// TIA Portal project "separating station" (V17)
// Vorlageprojekt für das Buch mit Zielsystem S7-1200

(* hardware
DEVICE "S7-1200-Station_1"  S7-1200 Station
   slot 0: "Baugruppenträger_0"  Rack  V1.0
   slot 1: "PLC_1"  CPU 1211C DC/DC/DC  6ES7 211-1AE40-0XB0  V4.1
*)

// ===== PLC "PLC_1"  CPU 1211C DC/DC/DC =====

VAR_GLOBAL   // PLC tag table "Standard-Variablentabelle"
   "senz 1" AT %I0.0 : Bool;
   "push 1 f" AT %I0.1 : Bool;
   "push 1 b" AT %I0.2 : Bool;
   "at push 1 exit" AT %I0.3 : Bool;
   "push 2 f" AT %I0.5 : Bool;
   "push 2 b" AT %I0.6 : Bool;
   "at push 2 exit" AT %I0.7 : Bool;
   "start" AT %I1.0 : Bool;
   "reset" AT %I1.1 : Bool;
   "stop" AT %I1.2 : Bool;
   "e stop" AT %I1.3 : Bool;
   "FACTORY io run" AT %I1.4 : Bool;
   "vs 1" AT %ID30 : DInt;
   "vs2" AT %ID34 : DInt;
   "entry conv 1" AT %Q0.0 : Bool;
   "pusher 1" AT %Q0.1 : Bool;
   "conv 1" AT %Q0.2 : Bool;
   "entry conv 2" AT %Q0.3 : Bool;
   "pusher 2" AT %Q0.4 : Bool;
   "conv 2" AT %Q0.5 : Bool;
   "start light" AT %Q0.6 : Bool;
   "reset light" AT %Q0.7 : Bool;
   "stop light" AT %Q1.0 : Bool;
   "count 2" AT %QD30 : DInt;
   "count 2(1)" AT %QD34 : DInt;
   "senz 2" AT %I0.4 : Bool;
   "temp" AT %MD30 : DInt;
   "Tag_1" AT %M0.1 : Bool;
   "Tag_2" AT %M0.2 : Bool;
   "Tag_3" AT %M0.3 : Bool;
   "Tag_4" AT %M0.4 : Bool;
   "Tag_5" AT %M0.5 : Bool;
   "Tag_6" AT %M0.6 : Bool;
   "Tag_7" AT %M0.7 : Bool;
   "Tag_8" AT %M1.0 : Bool;
   "Tag_9" AT %M1.1 : Bool;
   "Tag_10" AT %M1.2 : Bool;
   "Tag_11" AT %MD34 : DWord;
   "Tag_12" AT %MD38 : DWord;
END_VAR

DATA_BLOCK "modes"   // DB2
{ S7_Optimized_Access := 'TRUE' }
VERSION : 0.1
   VAR
      "stop mode" : Bool;
      "start mode" : Bool;
      "auto mode" : Bool;
      "reset mode" : Bool;
      "e stop mode" : Bool;
      "home position" : Bool;
   END_VAR
BEGIN
END_DATA_BLOCK

DATA_BLOCK "steps"   // DB4
{ S7_Optimized_Access := 'TRUE' }
VERSION : 0.1
   VAR
      "next step" : Int := 0;
      "curent step" : Int := 0;
   END_VAR
BEGIN
END_DATA_BLOCK

FUNCTION "1 operation modes" : Void   // FC1, LAD
{ S7_Optimized_Access := 'TRUE' }
VERSION : 0.1
BEGIN

REGION Network 1: start mode
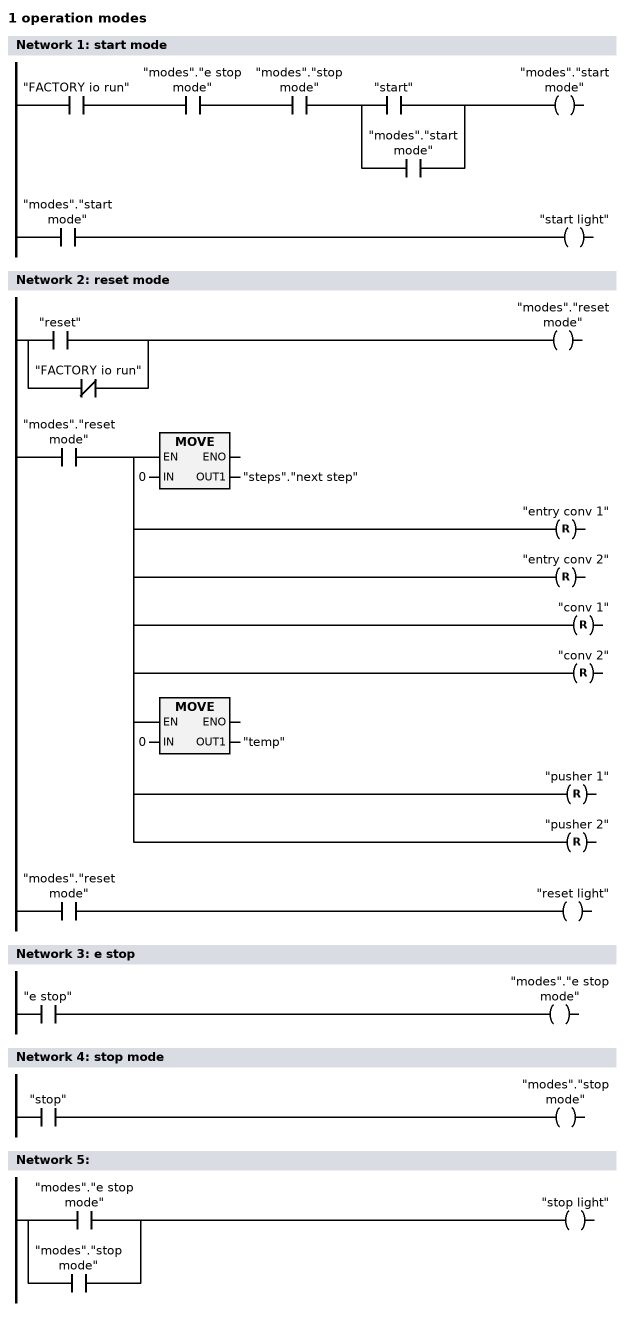
   RUNG wire#powerrail
      Contact( "FACTORY io run" )
      Contact( "modes"."e stop mode" )
      Contact( "modes"."stop mode" )
      wire#w1
      Contact( "start" )
      wire#w2
      Coil( "modes"."start mode" )
   END_RUNG
   RUNG wire#w1
      Contact( "modes"."start mode" )
   END_RUNG wire#w2
   RUNG wire#powerrail
      Contact( "modes"."start mode" )
      Coil( "start light" )
   END_RUNG
   // the same network as SCL:
   "modes"."start mode" := "FACTORY io run" AND "modes"."e stop mode" AND "modes"."stop mode" AND ("start" OR "modes"."start mode");
   "start light" := "modes"."start mode";
END_REGION

REGION Network 2: reset mode
   RUNG wire#powerrail
      Contact( "reset" )
      wire#w1
      Coil( "modes"."reset mode" )
   END_RUNG
   RUNG wire#powerrail
      I_Contact( "FACTORY io run" )
   END_RUNG wire#w1
   RUNG wire#powerrail
      Contact( "modes"."reset mode" )
      wire#w2
      Move(in := 0, out1 => "steps"."next step")
   END_RUNG
   RUNG wire#w2
      R_Coil( "entry conv 1" )
   END_RUNG
   RUNG wire#w2
      R_Coil( "entry conv 2" )
   END_RUNG
   RUNG wire#w2
      R_Coil( "conv 1" )
   END_RUNG
   RUNG wire#w2
      R_Coil( "conv 2" )
   END_RUNG
   RUNG wire#w2
      Move(in := 0, out1 => "temp")
   END_RUNG
   RUNG wire#w2
      R_Coil( "pusher 1" )
   END_RUNG
   RUNG wire#w2
      R_Coil( "pusher 2" )
   END_RUNG
   RUNG wire#powerrail
      Contact( "modes"."reset mode" )
      Coil( "reset light" )
   END_RUNG
   // the same network as SCL:
   "modes"."reset mode" := "reset" OR NOT "FACTORY io run";
   IF "modes"."reset mode" THEN
       "steps"."next step" := 0;
       "entry conv 1" := FALSE;
       "entry conv 2" := FALSE;
       "conv 1" := FALSE;
       "conv 2" := FALSE;
       "temp" := 0;
       "pusher 1" := FALSE;
       "pusher 2" := FALSE;
   END_IF;
   "reset light" := "modes"."reset mode";
END_REGION

REGION Network 3: e stop
   RUNG wire#powerrail
      Contact( "e stop" )
      Coil( "modes"."e stop mode" )
   END_RUNG
   // the same network as SCL:
   "modes"."e stop mode" := "e stop";
END_REGION

REGION Network 4: stop mode
   RUNG wire#powerrail
      Contact( "stop" )
      Coil( "modes"."stop mode" )
   END_RUNG
   // the same network as SCL:
   "modes"."stop mode" := "stop";
END_REGION

REGION Network 5
   RUNG wire#powerrail
      Contact( "modes"."e stop mode" )
      wire#w1
      Coil( "stop light" )
   END_RUNG
   RUNG wire#powerrail
      Contact( "modes"."stop mode" )
   END_RUNG wire#w1
   // the same network as SCL:
   "stop light" := "modes"."e stop mode" OR "modes"."stop mode";
END_REGION
END_FUNCTION

FUNCTION "2 step definition" : Void   // FC2, LAD
{ S7_Optimized_Access := 'TRUE' }
VERSION : 0.1
   VAR_TEMP   // added for the SCL form of the ladder/FBD networks
      _w1 : Bool;
   END_VAR
BEGIN

REGION Network 1
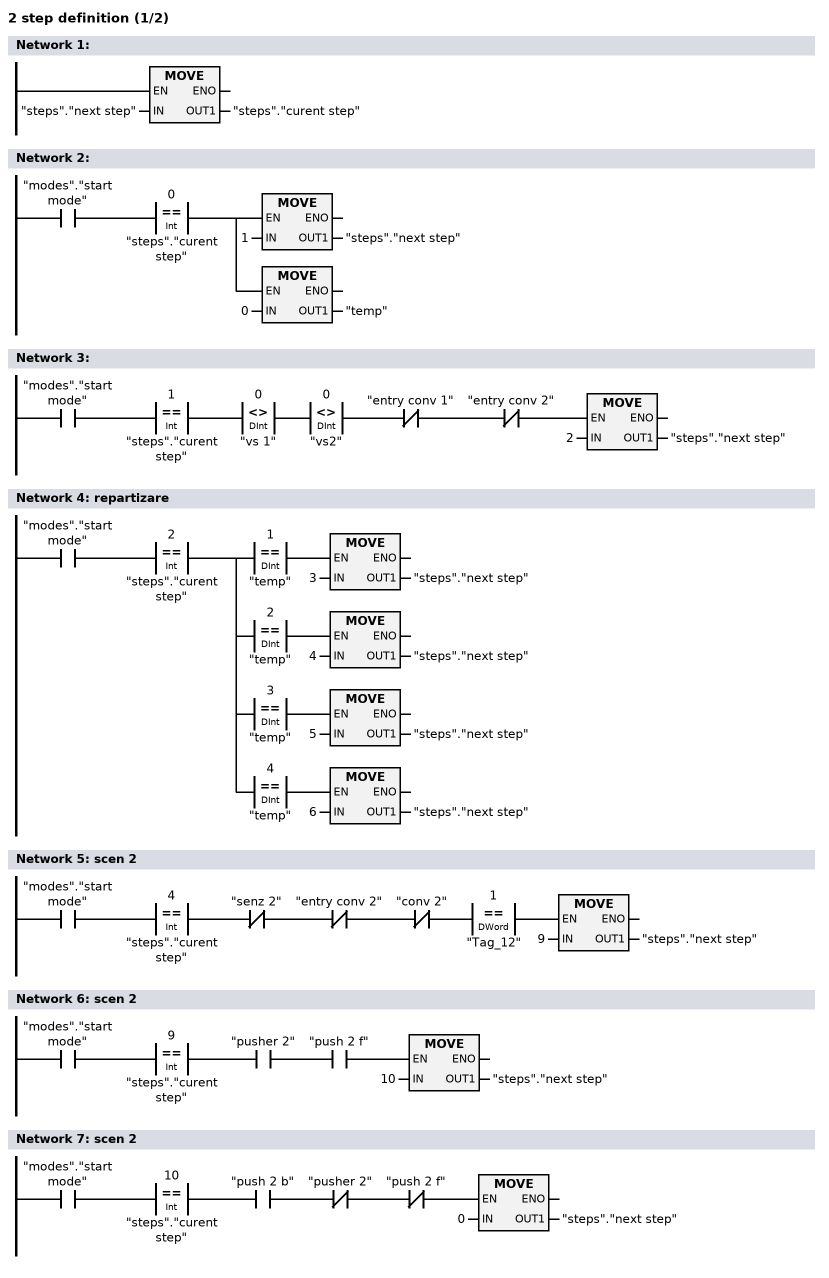
   RUNG wire#powerrail
      Move(in := "steps"."next step", out1 => "steps"."curent step")
   END_RUNG
   // the same network as SCL:
   "steps"."curent step" := "steps"."next step";
END_REGION

REGION Network 2
   RUNG wire#powerrail
      Contact( "modes"."start mode" )
      { S7_Templates := "SrcType := Int" } EQ_Contact(in1 := 0, in2 := "steps"."curent step")
      wire#w1
      Move(in := 1, out1 => "steps"."next step")
   END_RUNG
   RUNG wire#w1
      Move(in := 0, out1 => "temp")
   END_RUNG
   // the same network as SCL:
   IF "modes"."start mode" AND (0 = "steps"."curent step") THEN
       "steps"."next step" := 1;
       "temp" := 0;
   END_IF;
END_REGION

REGION Network 3
   RUNG wire#powerrail
      Contact( "modes"."start mode" )
      { S7_Templates := "SrcType := Int" } EQ_Contact(in1 := 1, in2 := "steps"."curent step")
      { S7_Templates := "SrcType := DInt" } NE_Contact(in1 := 0, in2 := "vs 1")
      { S7_Templates := "SrcType := DInt" } NE_Contact(in1 := 0, in2 := "vs2")
      I_Contact( "entry conv 1" )
      I_Contact( "entry conv 2" )
      Move(in := 2, out1 => "steps"."next step")
   END_RUNG
   // the same network as SCL:
   IF "modes"."start mode" AND (1 = "steps"."curent step") AND (0 <> "vs 1") AND (0 <> "vs2") AND NOT "entry conv 1" AND NOT "entry conv 2" THEN
       "steps"."next step" := 2;
   END_IF;
END_REGION

REGION Network 4: repartizare
   RUNG wire#powerrail
      Contact( "modes"."start mode" )
      { S7_Templates := "SrcType := Int" } EQ_Contact(in1 := 2, in2 := "steps"."curent step")
      wire#w1
      { S7_Templates := "SrcType := DInt" } EQ_Contact(in1 := 1, in2 := "temp")
      Move(in := 3, out1 => "steps"."next step")
   END_RUNG
   RUNG wire#w1
      { S7_Templates := "SrcType := DInt" } EQ_Contact(in1 := 2, in2 := "temp")
      Move(in := 4, out1 => "steps"."next step")
   END_RUNG
   RUNG wire#w1
      { S7_Templates := "SrcType := DInt" } EQ_Contact(in1 := 3, in2 := "temp")
      Move(in := 5, out1 => "steps"."next step")
   END_RUNG
   RUNG wire#w1
      { S7_Templates := "SrcType := DInt" } EQ_Contact(in1 := 4, in2 := "temp")
      Move(in := 6, out1 => "steps"."next step")
   END_RUNG
   // the same network as SCL:
   #_w1 := "modes"."start mode" AND (2 = "steps"."curent step");
   IF #_w1 AND (1 = "temp") THEN "steps"."next step" := 3; END_IF;
   IF #_w1 AND (2 = "temp") THEN "steps"."next step" := 4; END_IF;
   IF #_w1 AND (3 = "temp") THEN "steps"."next step" := 5; END_IF;
   IF #_w1 AND (4 = "temp") THEN "steps"."next step" := 6; END_IF;
END_REGION

REGION Network 5: scen 2
   RUNG wire#powerrail
      Contact( "modes"."start mode" )
      { S7_Templates := "SrcType := Int" } EQ_Contact(in1 := 4, in2 := "steps"."curent step")
      I_Contact( "senz 2" )
      I_Contact( "entry conv 2" )
      I_Contact( "conv 2" )
      { S7_Templates := "SrcType := DWord" } EQ_Contact(in1 := 1, in2 := "Tag_12")
      Move(in := 9, out1 => "steps"."next step")
   END_RUNG
   // the same network as SCL:
   IF "modes"."start mode" AND (4 = "steps"."curent step") AND NOT "senz 2" AND NOT "entry conv 2" AND NOT "conv 2" AND (1 = "Tag_12") THEN
       "steps"."next step" := 9;
   END_IF;
END_REGION

REGION Network 6: scen 2
   RUNG wire#powerrail
      Contact( "modes"."start mode" )
      { S7_Templates := "SrcType := Int" } EQ_Contact(in1 := 9, in2 := "steps"."curent step")
      Contact( "pusher 2" )
      Contact( "push 2 f" )
      Move(in := 10, out1 => "steps"."next step")
   END_RUNG
   // the same network as SCL:
   IF "modes"."start mode" AND (9 = "steps"."curent step") AND "pusher 2" AND "push 2 f" THEN
       "steps"."next step" := 10;
   END_IF;
END_REGION

REGION Network 7: scen 2
   RUNG wire#powerrail
      Contact( "modes"."start mode" )
      { S7_Templates := "SrcType := Int" } EQ_Contact(in1 := 10, in2 := "steps"."curent step")
      Contact( "push 2 b" )
      I_Contact( "pusher 2" )
      I_Contact( "push 2 f" )
      Move(in := 0, out1 => "steps"."next step")
   END_RUNG
   // the same network as SCL:
   IF "modes"."start mode" AND (10 = "steps"."curent step") AND "push 2 b" AND NOT "pusher 2" AND NOT "push 2 f" THEN
       "steps"."next step" := 0;
   END_IF;
END_REGION

REGION Network 8: scenariu 3
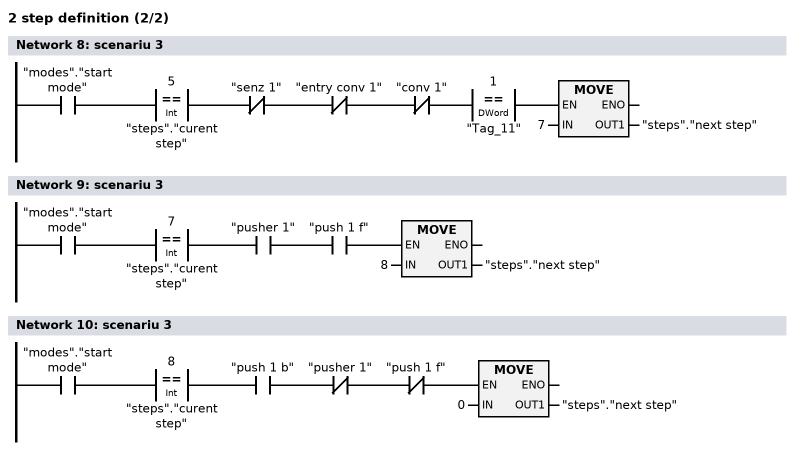
   RUNG wire#powerrail
      Contact( "modes"."start mode" )
      { S7_Templates := "SrcType := Int" } EQ_Contact(in1 := 5, in2 := "steps"."curent step")
      I_Contact( "senz 1" )
      I_Contact( "entry conv 1" )
      I_Contact( "conv 1" )
      { S7_Templates := "SrcType := DWord" } EQ_Contact(in1 := 1, in2 := "Tag_11")
      Move(in := 7, out1 => "steps"."next step")
   END_RUNG
   // the same network as SCL:
   IF "modes"."start mode" AND (5 = "steps"."curent step") AND NOT "senz 1" AND NOT "entry conv 1" AND NOT "conv 1" AND (1 = "Tag_11") THEN
       "steps"."next step" := 7;
   END_IF;
END_REGION

REGION Network 9: scenariu 3
   RUNG wire#powerrail
      Contact( "modes"."start mode" )
      { S7_Templates := "SrcType := Int" } EQ_Contact(in1 := 7, in2 := "steps"."curent step")
      Contact( "pusher 1" )
      Contact( "push 1 f" )
      Move(in := 8, out1 => "steps"."next step")
   END_RUNG
   // the same network as SCL:
   IF "modes"."start mode" AND (7 = "steps"."curent step") AND "pusher 1" AND "push 1 f" THEN
       "steps"."next step" := 8;
   END_IF;
END_REGION

REGION Network 10: scenariu 3
   RUNG wire#powerrail
      Contact( "modes"."start mode" )
      { S7_Templates := "SrcType := Int" } EQ_Contact(in1 := 8, in2 := "steps"."curent step")
      Contact( "push 1 b" )
      I_Contact( "pusher 1" )
      I_Contact( "push 1 f" )
      Move(in := 0, out1 => "steps"."next step")
   END_RUNG
   // the same network as SCL:
   IF "modes"."start mode" AND (8 = "steps"."curent step") AND "push 1 b" AND NOT "pusher 1" AND NOT "push 1 f" THEN
       "steps"."next step" := 0;
   END_IF;
END_REGION
END_FUNCTION

FUNCTION "3 step execution" : Void   // FC3, LAD
{ S7_Optimized_Access := 'TRUE' }
VERSION : 0.1
   VAR_TEMP   // added for the SCL form of the ladder/FBD networks
      _w1 : Bool;
      _w2 : Bool;
   END_VAR
BEGIN

REGION Network 1
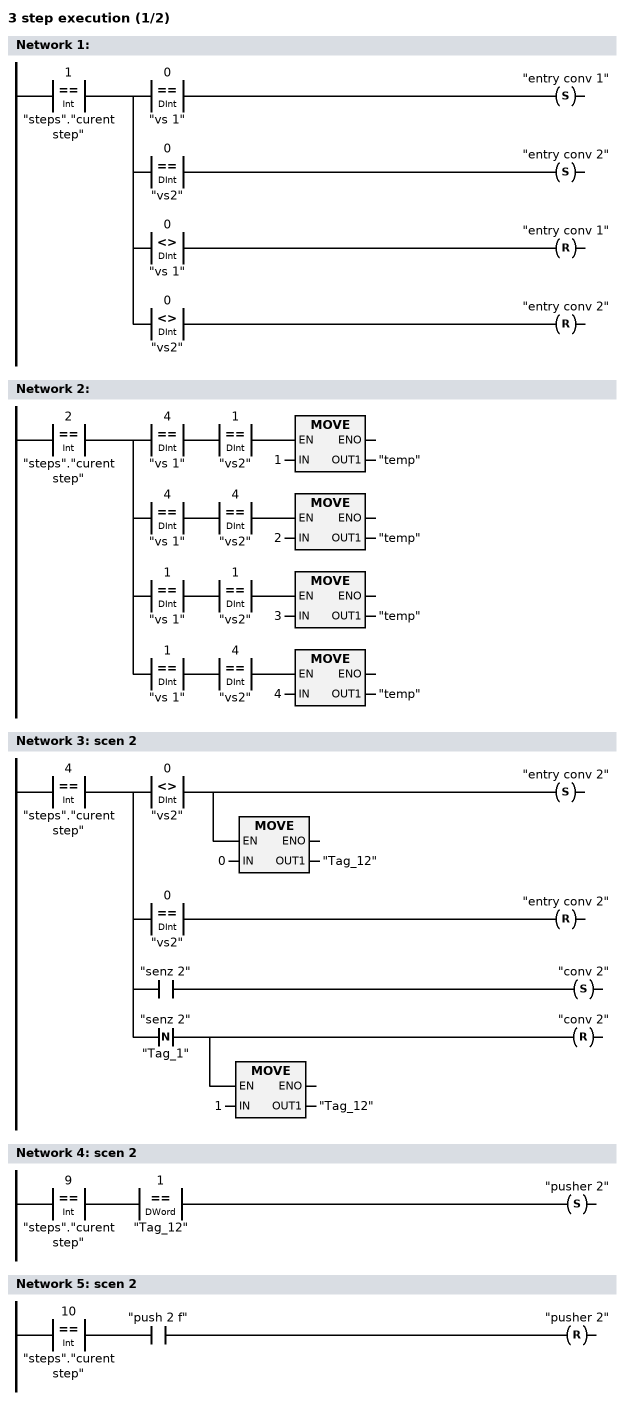
   RUNG wire#powerrail
      { S7_Templates := "SrcType := Int" } EQ_Contact(in1 := 1, in2 := "steps"."curent step")
      wire#w1
      { S7_Templates := "SrcType := DInt" } EQ_Contact(in1 := 0, in2 := "vs 1")
      S_Coil( "entry conv 1" )
   END_RUNG
   RUNG wire#w1
      { S7_Templates := "SrcType := DInt" } EQ_Contact(in1 := 0, in2 := "vs2")
      S_Coil( "entry conv 2" )
   END_RUNG
   RUNG wire#w1
      { S7_Templates := "SrcType := DInt" } NE_Contact(in1 := 0, in2 := "vs 1")
      R_Coil( "entry conv 1" )
   END_RUNG
   RUNG wire#w1
      { S7_Templates := "SrcType := DInt" } NE_Contact(in1 := 0, in2 := "vs2")
      R_Coil( "entry conv 2" )
   END_RUNG
   // the same network as SCL:
   #_w1 := 1 = "steps"."curent step";
   IF #_w1 AND (0 = "vs 1") THEN "entry conv 1" := TRUE; END_IF;
   IF #_w1 AND (0 = "vs2") THEN "entry conv 2" := TRUE; END_IF;
   IF #_w1 AND (0 <> "vs 1") THEN "entry conv 1" := FALSE; END_IF;
   IF #_w1 AND (0 <> "vs2") THEN "entry conv 2" := FALSE; END_IF;
END_REGION

REGION Network 2
   RUNG wire#powerrail
      { S7_Templates := "SrcType := Int" } EQ_Contact(in1 := 2, in2 := "steps"."curent step")
      wire#w1
      { S7_Templates := "SrcType := DInt" } EQ_Contact(in1 := 4, in2 := "vs 1")
      { S7_Templates := "SrcType := DInt" } EQ_Contact(in1 := 1, in2 := "vs2")
      Move(in := 1, out1 => "temp")
   END_RUNG
   RUNG wire#w1
      { S7_Templates := "SrcType := DInt" } EQ_Contact(in1 := 4, in2 := "vs 1")
      { S7_Templates := "SrcType := DInt" } EQ_Contact(in1 := 4, in2 := "vs2")
      Move(in := 2, out1 => "temp")
   END_RUNG
   RUNG wire#w1
      { S7_Templates := "SrcType := DInt" } EQ_Contact(in1 := 1, in2 := "vs 1")
      { S7_Templates := "SrcType := DInt" } EQ_Contact(in1 := 1, in2 := "vs2")
      Move(in := 3, out1 => "temp")
   END_RUNG
   RUNG wire#w1
      { S7_Templates := "SrcType := DInt" } EQ_Contact(in1 := 1, in2 := "vs 1")
      { S7_Templates := "SrcType := DInt" } EQ_Contact(in1 := 4, in2 := "vs2")
      Move(in := 4, out1 => "temp")
   END_RUNG
   // the same network as SCL:
   #_w1 := 2 = "steps"."curent step";
   IF #_w1 AND (4 = "vs 1") AND (1 = "vs2") THEN "temp" := 1; END_IF;
   IF #_w1 AND (4 = "vs 1") AND (4 = "vs2") THEN "temp" := 2; END_IF;
   IF #_w1 AND (1 = "vs 1") AND (1 = "vs2") THEN "temp" := 3; END_IF;
   IF #_w1 AND (1 = "vs 1") AND (4 = "vs2") THEN "temp" := 4; END_IF;
END_REGION

REGION Network 3: scen 2
   RUNG wire#powerrail
      { S7_Templates := "SrcType := Int" } EQ_Contact(in1 := 4, in2 := "steps"."curent step")
      wire#w1
      { S7_Templates := "SrcType := DInt" } NE_Contact(in1 := 0, in2 := "vs2")
      wire#w2
      S_Coil( "entry conv 2" )
   END_RUNG
   RUNG wire#w2
      Move(in := 0, out1 => "Tag_12")
   END_RUNG
   RUNG wire#w1
      { S7_Templates := "SrcType := DInt" } EQ_Contact(in1 := 0, in2 := "vs2")
      R_Coil( "entry conv 2" )
   END_RUNG
   RUNG wire#w1
      Contact( "senz 2" )
      S_Coil( "conv 2" )
   END_RUNG
   RUNG wire#w1
      N_Contact(operand := "senz 2", bit := "Tag_1")
      wire#w3
      R_Coil( "conv 2" )
   END_RUNG
   RUNG wire#w3
      Move(in := 1, out1 => "Tag_12")
   END_RUNG
   // the same network as SCL:
   #_w1 := 4 = "steps"."curent step";
   IF #_w1 AND (0 <> "vs2") THEN
       "entry conv 2" := TRUE;
       "Tag_12" := 0;
   END_IF;
   IF #_w1 AND (0 = "vs2") THEN "entry conv 2" := FALSE; END_IF;
   IF #_w1 AND "senz 2" THEN "conv 2" := TRUE; END_IF;
   #_w2 := #_w1 AND NOT "senz 2" AND "Tag_1";   // falling edge of "senz 2"
   "Tag_1" := "senz 2";
   IF #_w2 THEN
       "conv 2" := FALSE;
       "Tag_12" := 1;
   END_IF;
END_REGION

REGION Network 4: scen 2
   RUNG wire#powerrail
      { S7_Templates := "SrcType := Int" } EQ_Contact(in1 := 9, in2 := "steps"."curent step")
      { S7_Templates := "SrcType := DWord" } EQ_Contact(in1 := 1, in2 := "Tag_12")
      S_Coil( "pusher 2" )
   END_RUNG
   // the same network as SCL:
   IF (9 = "steps"."curent step") AND (1 = "Tag_12") THEN "pusher 2" := TRUE; END_IF;
END_REGION

REGION Network 5: scen 2
   RUNG wire#powerrail
      { S7_Templates := "SrcType := Int" } EQ_Contact(in1 := 10, in2 := "steps"."curent step")
      Contact( "push 2 f" )
      R_Coil( "pusher 2" )
   END_RUNG
   // the same network as SCL:
   IF (10 = "steps"."curent step") AND "push 2 f" THEN "pusher 2" := FALSE; END_IF;
END_REGION

REGION Network 6: scen 3
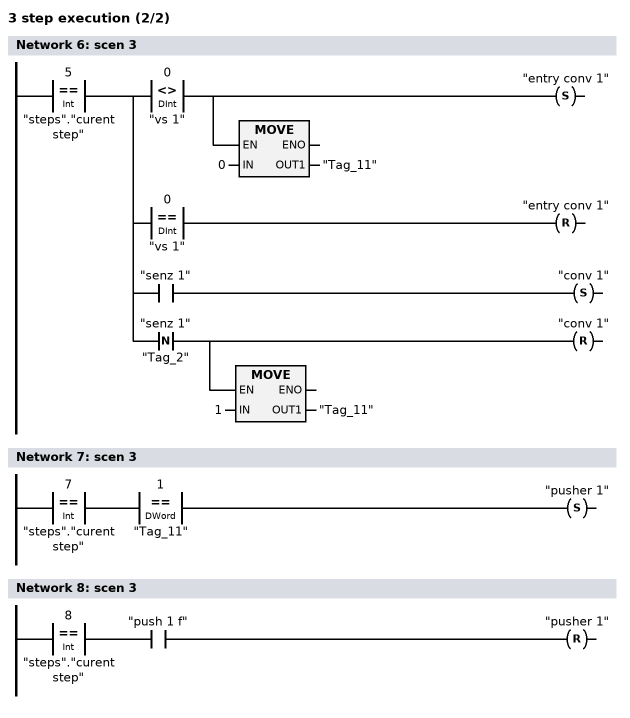
   RUNG wire#powerrail
      { S7_Templates := "SrcType := Int" } EQ_Contact(in1 := 5, in2 := "steps"."curent step")
      wire#w1
      { S7_Templates := "SrcType := DInt" } NE_Contact(in1 := 0, in2 := "vs 1")
      wire#w2
      S_Coil( "entry conv 1" )
   END_RUNG
   RUNG wire#w2
      Move(in := 0, out1 => "Tag_11")
   END_RUNG
   RUNG wire#w1
      { S7_Templates := "SrcType := DInt" } EQ_Contact(in1 := 0, in2 := "vs 1")
      R_Coil( "entry conv 1" )
   END_RUNG
   RUNG wire#w1
      Contact( "senz 1" )
      S_Coil( "conv 1" )
   END_RUNG
   RUNG wire#w1
      N_Contact(operand := "senz 1", bit := "Tag_2")
      wire#w3
      R_Coil( "conv 1" )
   END_RUNG
   RUNG wire#w3
      Move(in := 1, out1 => "Tag_11")
   END_RUNG
   // the same network as SCL:
   #_w1 := 5 = "steps"."curent step";
   IF #_w1 AND (0 <> "vs 1") THEN
       "entry conv 1" := TRUE;
       "Tag_11" := 0;
   END_IF;
   IF #_w1 AND (0 = "vs 1") THEN "entry conv 1" := FALSE; END_IF;
   IF #_w1 AND "senz 1" THEN "conv 1" := TRUE; END_IF;
   #_w2 := #_w1 AND NOT "senz 1" AND "Tag_2";   // falling edge of "senz 1"
   "Tag_2" := "senz 1";
   IF #_w2 THEN
       "conv 1" := FALSE;
       "Tag_11" := 1;
   END_IF;
END_REGION

REGION Network 7: scen 3
   RUNG wire#powerrail
      { S7_Templates := "SrcType := Int" } EQ_Contact(in1 := 7, in2 := "steps"."curent step")
      { S7_Templates := "SrcType := DWord" } EQ_Contact(in1 := 1, in2 := "Tag_11")
      S_Coil( "pusher 1" )
   END_RUNG
   // the same network as SCL:
   IF (7 = "steps"."curent step") AND (1 = "Tag_11") THEN "pusher 1" := TRUE; END_IF;
END_REGION

REGION Network 8: scen 3
   RUNG wire#powerrail
      { S7_Templates := "SrcType := Int" } EQ_Contact(in1 := 8, in2 := "steps"."curent step")
      Contact( "push 1 f" )
      R_Coil( "pusher 1" )
   END_RUNG
   // the same network as SCL:
   IF (8 = "steps"."curent step") AND "push 1 f" THEN "pusher 1" := FALSE; END_IF;
END_REGION
END_FUNCTION

FUNCTION "MHJ-PLC-Lab-Function-S71200" : Void   // FC9000, SCL
{ S7_Optimized_Access := 'TRUE' }
VERSION : 0.1
   VAR_TEMP
      rdTimeReturn : Int;
      outputTime : DTL;
      SyncVal : Byte;
      forVal : Int;
      forVal_2 : Int;
      Value : Byte;
   END_VAR
   VAR CONSTANT
      CompVal : Byte := 16#34;
      Value_01 : Byte := 16#11;
      Value_01_DW : DWord := 16#A165_D992;
      Value_02_DW : DWord := 16#58BE_4401;
   END_VAR
BEGIN

   #Value:=PEEK(area := 16#82,
        dbNumber := 0,
        byteOffset := 511);
   #Value := #Value + 1;

   POKE(area := 16#82,
        dbNumber := 0,
        byteOffset := 511,
        value := #Value);

   POKE(area:=16#81,
        dbNumber:=0,
        byteOffset:=1016,
        value:=#Value_01_DW);
   POKE(area := 16#81,
        dbNumber := 0,
        byteOffset := 1020,
        value := #Value_02_DW);

   POKE(area := 16#81,
        dbNumber := 0,
        byteOffset := 511,
        value := B#16#00);

   FOR #forVal := 0 TO 120 DO
       FOR #forVal_2:=0 TO 10 DO
           #rdTimeReturn:=RD_SYS_T(#outputTime);
           #rdTimeReturn := WR_SYS_T(#outputTime);
           #rdTimeReturn := RD_SYS_T(#outputTime);
           #rdTimeReturn := WR_SYS_T(#outputTime);
       END_FOR;
       #SyncVal:= PEEK(area := 16#81,
                      dbNumber := 0,
                      byteOffset := 511);
       IF #SyncVal = #CompVal THEN
          GOTO M_1;
       END_IF;
   END_FOR;
   RETURN;

   M_1:
   POKE(area := 16#81,
        dbNumber := 0,
        byteOffset := 511,
        value := B#16#0);
END_FUNCTION

ORGANIZATION_BLOCK "Main"   // OB1, FBD, ProgramCycle
TITLE = "Main Program Sweep (Cycle)"
{ S7_Optimized_Access := 'TRUE' }
VERSION : 0.1
   VAR_INPUT
      Initial_Call : Bool;   // Initial call of this OB
      Remanence : Bool;   // =True, if remanent data are available
   END_VAR
BEGIN

REGION Network 1: Konnektierungsbaustein für PLC-Lab
   // Im Netzwerk 1 wird der Konnektierungsbaustein für PLC-Lab aufgerufen.
   // Dieser Aufruf darf nicht entfernt werden!
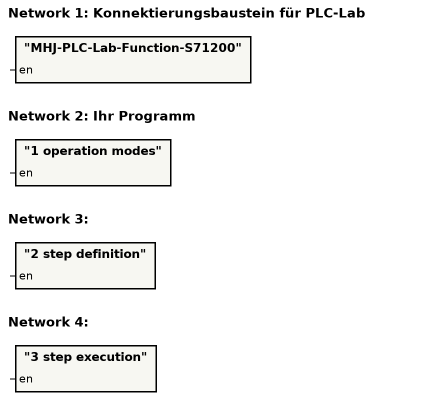
   "MHJ-PLC-Lab-Function-S71200"();
END_REGION

REGION Network 2: Ihr Programm
   // Schreiben Sie ab Netzwerk 2 Ihr Programm
   "1 operation modes"();
END_REGION

REGION Network 3
   "2 step definition"();
END_REGION

REGION Network 4
   "3 step execution"();
END_REGION
END_ORGANIZATION_BLOCK